(* CoDeSys 2.3.9.52 project: TrafficLights_pedeX_v1_Template.pro *)
(* Libraries: STANDARD.LIB*16.8.17 14:08:57 *)

(* Global variable list: Global_Variables *)
VAR_GLOBAL
	I_S1		: BOOL; (*Pedestrian X button North*)
	I_S2		: BOOL; (*Pedestrian X button South*)
	O_L1_N_Red	: BOOL; (*Light red, Pedestrian North-South*)
	O_L3_N_Grn	: BOOL;	(*Light green, Pedestrian North-South*)
	O_L4_E_Red	: BOOL;	(*Light red, Cars East-West*)
	O_L5_E_Yel	: BOOL;	(*Light yellow, Cars East-West*)
	O_L6_E_Grn	: BOOL;	(*Light green, Cars East-West*)
END_VAR

(* POU PRG_BlinkingSimple, ST *)
PROGRAM PRG_BlinkingSimple
(*Niko Siltala
Avustavia laskentaoperaatioita
- vilkutussignaalit
*)
VAR_OUTPUT
	bSign1Hz:BOOL;					(*1 Hz (60krt/min) taajudella vaihteleva signaali*)
END_VAR
VAR
	bInitDone	: BOOL	:=FALSE;	(*Ohjelman initialisointi*)
	c : INT	:=0;				(*Blink counter*)
END_VAR
(*Ohjelman initialisoinnit - Suoritetaan vain kertaalleen*)
IF NOT bInitDone THEN
	bInitDone := TRUE;
END_IF;

(*Making 1Hz blinking signal in case of simulator*)
CASE c OF
0:
	bSign1Hz:= TRUE;
1:
	bSign1Hz:= FALSE;
ELSE
	bSign1Hz:= FALSE;
END_CASE;

(*Add counter *)
c:= c + 1;
IF c > 1 THEN
	c := 0;
END_IF;
END_PROGRAM

(* POU SFC_StateModel, SFC *)
PROGRAM SFC_StateModel
VAR
	tDelay	: TIME	:= T#2s;
	tDelay_Walk : TIME := T#5s;
END_VAR
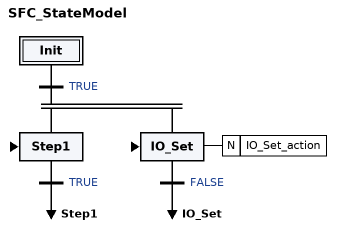
INITIAL_STEP Init:
END_STEP
TRANSITION FROM Init TO (Step1, IO_Set) := TRUE;
END_TRANSITION
STEP Step1:
END_STEP
TRANSITION FROM Step1 TO Step1 := TRUE;
END_TRANSITION
STEP IO_Set:
	IO_Set_action(N);
END_STEP
TRANSITION FROM IO_Set TO IO_Set := FALSE;
END_TRANSITION

ACTION IO_Set_action:
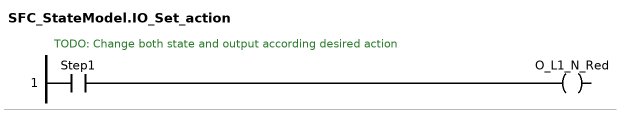
_LD_ (* Ladder Diagram *)
NETWORK 1 (* TODO: Change both state and output according desired action *)
	[Step1] --- (O_L1_N_Red)
_END_LD_
(* the same logic as Structured Text *)
(* Network 1: TODO: Change both state and output according desired action *)
O_L1_N_Red := Step1;
END_ACTION
END_PROGRAM

(* Visualisation VC_Main
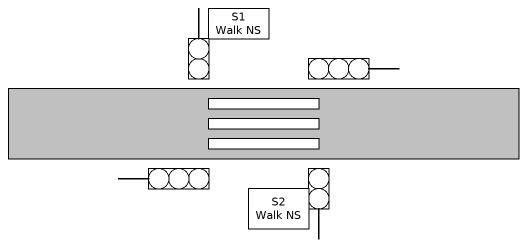
ellipse at (300,160)-(321,181): alarm colour if .O_L1_N_Red
ellipse at (300,180)-(321,201): alarm colour if .O_L3_N_Grn
rounded rectangle at (200,0)-(261,31): text "S1 / Walk NS"; alarm colour if .I_S1; taps .I_S1
rounded rectangle at (240,180)-(301,221): text "S2 / Walk NS"; alarm colour if .I_S2; taps .I_S2
ellipse at (180,160)-(201,181): alarm colour if .O_L4_E_Red
ellipse at (160,160)-(181,181): alarm colour if .O_L5_E_Yel
ellipse at (140,160)-(161,181): alarm colour if .O_L6_E_Grn
ellipse at (300,50)-(321,71): alarm colour if .O_L4_E_Red
ellipse at (320,50)-(341,71): alarm colour if .O_L5_E_Yel
ellipse at (340,50)-(361,71): alarm colour if .O_L6_E_Grn
ellipse at (180,50)-(201,71): alarm colour if .O_L1_N_Red
ellipse at (180,30)-(201,51): alarm colour if .O_L3_N_Grn
12 more shapes without text or variables
*)
